{attribute 'qualified_only'}
VAR_GLOBAL
	
	//Recipe Parameters from HMI
	stInfo			: ST_RecipeInfo;			// info Parameters
	stSolventNTimes	: ST_RecipeSolventAndTimes;	// Solvent and Times Parameters
	stVolumes		: ST_RecipeVolumes;			// Volumes Parameters
	stOtherParams	: ST_RecipeOtherParams;		// Other Parameters
	stFileInfo		: ST_RecipeFileInfo;		// Json file info
	
	stCurrentRecipe : ST_Recipe; // Used by HMI and active cycle
    stActiveRecipe  : ST_Recipe; // Applied in the process
	
	sSelectedRecipeName	: STRING(256); //Json filename 
	
	//aAvailableFiles : ARRAY[0..49] OF ST_RecipeFileInfo; // Recipe folder files
    //iFileCount      : INT;
	
	bIsThereRecipeActivated	: BOOL := FALSE; //Flag to identify if there is a recipe activated before start the autocycle. 	
	
END_VAR

(* stored: Version 1.1.0.1, ProductVersion 3.1.4024.15
   GVL GVL_Recipe: Id {dea22a66-1424-457b-bb31-9cb7538a2d73} *)
